KUKA KRL program: chk_w5_grp1_vacoff.src

&ACCESS RV
&COMMENT Actros Vaccum off
DEF chk_w5_grp1_vacoff( )

; Check Vacuum on gripper ACTROS
;//---- Start User-------

$TIMER[10] = 0
$TIMER_STOP[10] = FALSE

WAIT FOR (NOT $IN[5])

$TIMER_STOP[10] = TRUE
$TIMER[10] = 0

;//---- End User---------

END
